// TIA Portal V16 export
// export: Created 2022-07-21T09:35:16.5415874Z, ExportSetting WithDefaults, DisplayName Totally Integrated Automation Portal, DisplayVersion V16 Update 4, DisplayName TIA Portal Version Control Interface, DisplayVersion V16 Update 2, DisplayName TIA Portal Openness, DisplayVersion V16 Update 4, DisplayName SINAMICS Startdrive Advanced, DisplayVersion V16 Update 5, DisplayName SINAMICS Startdrive G130, G150, S120, S150, SINAMICS MV, S210, DisplayVersion V16 Update 5, DisplayName SINAMICS Startdrive G110M, G120, G120C, G120D, G120P, G115D, DisplayVersion V16 Update 5, DisplayName STEP 7 Professional, DisplayVersion V16 Update 4, DisplayName STEP 7 Safety, DisplayVersion V16, DisplayName WinCC Advanced, DisplayVersion V16 Update 4
FUNCTION_BLOCK "fbIDReadingCognexHand"   // FB27, LAD
TITLE = Cognex camera / Obsługa kamery Cognex
{ S7_Optimized_Access := 'TRUE' }
VERSION : 0.1
// stored: AutoNumber false, IsIECCheckEnabled true, IsRetainMemResEnabled false, MemoryReserve 100, SetENOAutomatically false, UDAEnableTagReadback false
   VAR_INPUT
      enableDevice { ExternalAccessible := 'False'; ExternalVisible := 'False'; ExternalWritable := 'False'} : Bool;   // Zezwolenie / Permission
      timeBootUp { ExternalAccessible := 'False'; ExternalVisible := 'False'; ExternalWritable := 'False'} : Time := T#5s;   // Czas uruchamiania kamery / Time boot up
      barcodeLength : Int;   // Długość barcode / Barcode length
      resultRightAlligned : Bool;   // Dopasowanie barcode do strony lewa/prawa / Barcode allign
      inCamera { ExternalAccessible := 'False'; ExternalVisible := 'False'; ExternalWritable := 'False'} : "typeIDReadingInputsCognex";   // Wejścia z kamery Cognex / Inputs camera Cognex
   END_VAR
   VAR_OUTPUT
      outCamera { ExternalAccessible := 'False'; ExternalVisible := 'False'; ExternalWritable := 'False'} : "typeIDReadingOutputsCognex";   // Wyjścia do kamery Cognex / Outputs camera Cognex
   END_VAR
   VAR_IN_OUT
      data : "typeCognex";   // Dane HMI Cognex / HMI Cognex data
   END_VAR
   VAR
      instGetInstancePath { ExternalAccessible := 'False'; ExternalVisible := 'False'; ExternalWritable := 'False'; S7_SetPoint := 'True'} : "fbGetInstancePath";
      sInstancePath { ExternalAccessible := 'False'; ExternalVisible := 'False'; ExternalWritable := 'False'} : String[100];
      statMemREResultAvailable { ExternalAccessible := 'False'; ExternalVisible := 'False'; ExternalWritable := 'False'} : Bool;   // Rezultat dostępny flaga pomocnicza / Result available memory
      statAmountofChars { ExternalAccessible := 'False'; ExternalVisible := 'False'; ExternalWritable := 'False'} : UInt;   // Liczba odczytanych znaków / Amount of characters read
      instMessageErrorDevice { ExternalAccessible := 'False'; ExternalVisible := 'False'; ExternalWritable := 'False'; S7_SetPoint := 'True'} : "fbMessageError";
      instMessageRate { ExternalAccessible := 'False'; ExternalVisible := 'False'; ExternalWritable := 'False'; S7_SetPoint := 'True'} : "fbMessageHandlingRate";
      instTOnBootUpDevice { ExternalAccessible := 'False'; ExternalVisible := 'False'; ExternalWritable := 'False'; S7_SetPoint := 'True'} : TON_TIME;
      sBootUpCompleteDevice { ExternalAccessible := 'False'; ExternalVisible := 'False'; ExternalWritable := 'False'} : Bool;
   END_VAR
   VAR_TEMP
      tDiff : Int;
      tAddString : String;
      tEnableDeviceMessages : Bool;
   END_VAR
   VAR CONSTANT
      constFiller : Char := '_';
      constNoRead : Char := '?';
      constInvalidData : Char := '!';
      constNoData : Char := '0';
      constRateWarning : Real := 50.0;
      constRateError : Real := 50.0;
      constAmountTillMessage : USInt := 5;
   END_VAR
   VAR_TEMP   // added for the SCL form of the ladder/FBD networks
      _w1 : Bool;
   END_VAR
BEGIN

REGION Network 1: Call: fbGetInstancePath / Wywołanie: fbGetInstancePath
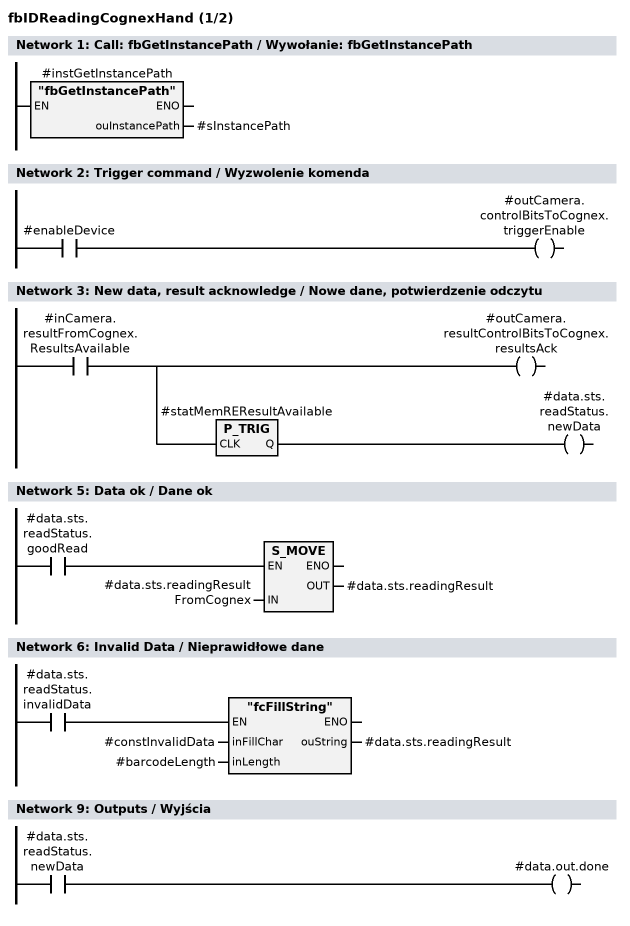
   RUNG wire#powerrail
      #instGetInstancePath(ouInstancePath => #sInstancePath)
   END_RUNG
   // the same network as SCL:
   #instGetInstancePath(ouInstancePath => #sInstancePath);   // "fbGetInstancePath"
END_REGION

REGION Network 2: Trigger command / Wyzwolenie komenda
   RUNG wire#powerrail
      Contact( #enableDevice )
      Coil( #outCamera.controlBitsToCognex.triggerEnable )
   END_RUNG
   // the same network as SCL:
   #outCamera.controlBitsToCognex.triggerEnable := #enableDevice;
END_REGION

REGION Network 3: New data, result acknowledge / Nowe dane, potwierdzenie odczytu
   RUNG wire#powerrail
      Contact( #inCamera.resultFromCognex.ResultsAvailable )
      wire#w1
      Coil( #outCamera.resultControlBitsToCognex.resultsAck )
   END_RUNG
   RUNG wire#w1
      P_Trig( #statMemREResultAvailable )
      Coil( #data.sts.readStatus.newData )
   END_RUNG
   // the same network as SCL:
   #outCamera.resultControlBitsToCognex.resultsAck := #inCamera.resultFromCognex.ResultsAvailable;
   #_w1 := #inCamera.resultFromCognex.ResultsAvailable AND NOT #statMemREResultAvailable;   // rising edge
   #statMemREResultAvailable := #inCamera.resultFromCognex.ResultsAvailable;
   #data.sts.readStatus.newData := #_w1;
END_REGION

REGION Network 4 (SCL): Process new data / Nowe dane - do obróbki

   // setting for readStatus and readingResultFromCognex (no output yet, only to evaluate !)
   IF #data.sts.readStatus.newData THEN

       #data.sts.readStatus.goodRead := FALSE;
       #data.sts.readStatus.invalidData := FALSE;

       #statAmountofChars := WORD_TO_UINT(#inCamera.resultDataFromCognex.ResultLength);

       // Get reading status
       IF #inCamera.resultDataFromCognex.GoodRead THEN
           REGION Good Read            
               #data.sts.readStatus.goodRead := TRUE;
               // Copy barcode
               Chars_TO_Strg(Chars := #inCamera.resultDataFromCognex.inspectionResults,
                             pChars := 0,
                             Cnt := #statAmountofChars,
                             Strg => #data.sts.readingResultFromCognex);
           END_REGION
       ELSIF  #inCamera.resultFromCognex.GeneralFault=TRUE THEN
           REGION Invalid Data
               #data.sts.readStatus.invalidData := TRUE;
               // Copy barcode
               Chars_TO_Strg(Chars := #inCamera.resultDataFromCognex.inspectionResults,
                             pChars := 0,
                             Cnt := #statAmountofChars,
                             Strg => #data.sts.readingResultFromCognex);

           END_REGION
       END_IF;
   END_IF;
END_REGION

REGION Network 5: Data ok / Dane ok
   RUNG wire#powerrail
      Contact( #data.sts.readStatus.goodRead )
      { S7_GenerateENO := "TRUE" } S_Move(in := #data.sts.readingResultFromCognex, out => #data.sts.readingResult)
   END_RUNG
   // the same network as SCL:
   IF #data.sts.readStatus.goodRead THEN
       #data.sts.readingResult := #data.sts.readingResultFromCognex;
   END_IF;
END_REGION

REGION Network 6: Invalid Data / Nieprawidłowe dane
   RUNG wire#powerrail
      Contact( #data.sts.readStatus.invalidData )
      "fcFillString"(inFillChar := #constInvalidData, inLength := #barcodeLength, ouString => #data.sts.readingResult)
   END_RUNG
   // the same network as SCL:
   IF #data.sts.readStatus.invalidData THEN
       "fcFillString"(inFillChar := #constInvalidData,
                      inLength := #barcodeLength,
                      ouString => #data.sts.readingResult);
   END_IF;
END_REGION

REGION Network 7 (SCL): Data ok - supplement data / Dane ok - uzupełnienie informacji

   //max length - max string length 
   #tDiff := #barcodeLength - LEN(#data.sts.readingResult);

   // check if reading result is long enough
   IF #tDiff <> 0 AND #data.sts.readStatus.goodRead THEN
     // build string to add to reading result
     #tAddString := '';
     FOR #tDiff := #tDiff TO 1 BY -1 DO
         #tAddString := CONCAT(IN1 := #tAddString, IN2 := #constFiller);
     END_FOR;
     // add string to reading result either as prefix or suffix
     IF #resultRightAlligned THEN
         #data.sts.readingResult := CONCAT(IN1:=#tAddString,IN2:=#data.sts.readingResult);
     ELSE
         #data.sts.readingResult := CONCAT(IN1:=#data.sts.readingResult,IN2:=#tAddString);
     END_IF;
   END_IF;
END_REGION

REGION Network 8 (SCL): Akceptuj numer LOT użytkownika
   IF #data.rq.acceptUserLOT THEN
       #data.sts.readingResult := #data.rq.userLOT;
   END_IF;
END_REGION

REGION Network 9: Outputs / Wyjścia
   RUNG wire#powerrail
      Contact( #data.sts.readStatus.newData )
      Coil( #data.out.done )
   END_RUNG
   // the same network as SCL:
   #data.out.done := #data.sts.readStatus.newData;
END_REGION

REGION Network 10: Messeges / Obsługa błędów
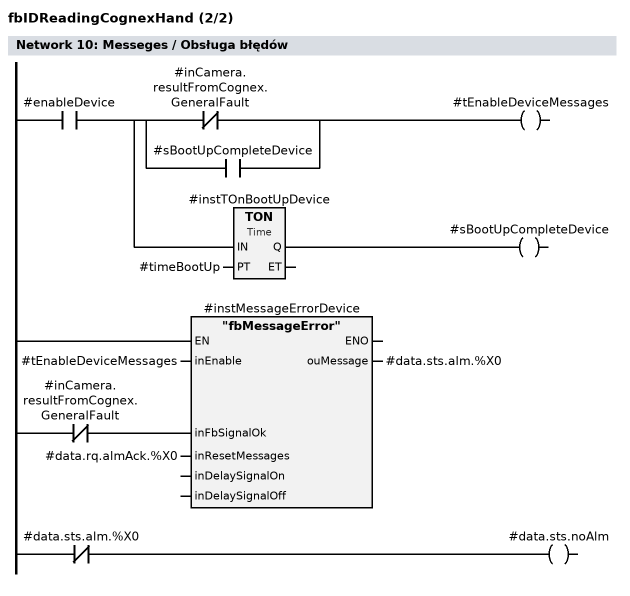
   RUNG wire#powerrail
      Contact( #enableDevice )
      wire#w1
      I_Contact( #inCamera.resultFromCognex.GeneralFault )
      wire#w2
      Coil( #tEnableDeviceMessages )
   END_RUNG
   RUNG wire#w1
      Contact( #sBootUpCompleteDevice )
   END_RUNG wire#w2
   RUNG wire#w1
      { S7_Templates := "time_type := Time" } #instTOnBootUpDevice.TON(pt := #timeBootUp, et =>)
      Coil( #sBootUpCompleteDevice )
   END_RUNG
   RUNG wire#powerrail
      #instMessageErrorDevice(inFbSignalOk := wire#w3, inEnable := #tEnableDeviceMessages, inResetMessages := #data.rq.almAck.%X0, inDelaySignalOn :=, inDelaySignalOff :=, ouMessage => #data.sts.alm.%X0)
   END_RUNG
   RUNG wire#powerrail
      I_Contact( #inCamera.resultFromCognex.GeneralFault )
   END_RUNG wire#w3
   RUNG wire#powerrail
      I_Contact( #data.sts.alm.%X0 )
      Coil( #data.sts.noAlm )
   END_RUNG
   // the same network as SCL:
   #tEnableDeviceMessages := #enableDevice AND (NOT #inCamera.resultFromCognex.GeneralFault OR #sBootUpCompleteDevice);
   #instTOnBootUpDevice(IN := #enableDevice, PT := #timeBootUp);   // TON
   #sBootUpCompleteDevice := #instTOnBootUpDevice.Q;
   #instMessageErrorDevice(inEnable := #tEnableDeviceMessages,   // "fbMessageError"
                           inFbSignalOk := NOT #inCamera.resultFromCognex.GeneralFault,
                           inResetMessages := #data.rq.almAck.%X0,
                           ouMessage => #data.sts.alm.%X0);
   #data.sts.noAlm := NOT #data.sts.alm.%X0;
END_REGION
END_FUNCTION_BLOCK
